PROGRAM main
VAR_INPUT
	X0 : bool;
	X1 : bool;
	X4 : bool;
	X5 : bool;
END_VAR

VAR_OUTPUT
	Y0 : bool;
END_VAR

VAR
	Y1 : bool;
END_VAR

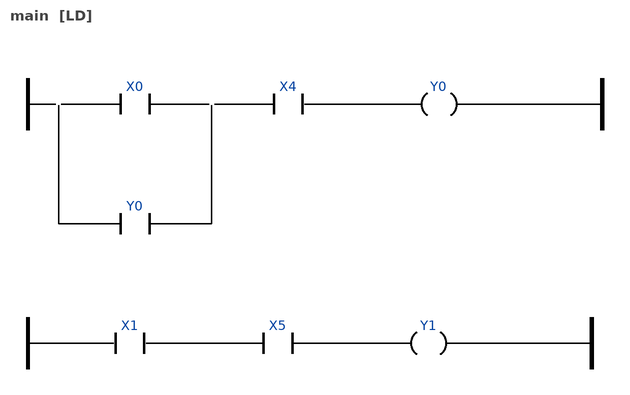
(* LD diagram, written out as Structured Text *)
Y0 := (Y0 OR X0) AND X4;
Y1 := X1 AND X5;
END_PROGRAM
